Fanuc KAREL source: MP0112.compact.KL

PROGRAM MP0112
%STACKSIZE=65535
%PRIORITY=65535
%NOLOCKGROUP
ROUTINE FINT(P1 : INTEGER) : INTEGER FROM MP0112
ROUTINE FREAL(P1 : REAL) : REAL FROM MP0112
ROUTINE RTEST(P1 : INTEGER; P2 : REAL) FROM MP0112
ROUTINE FINT
BEGIN
RETURN((P1 + 1))
END FINT
ROUTINE FREAL
BEGIN
RETURN((P1 + 1.0))
END FREAL
ROUTINE RTEST
VAR
L1 : XYZWPR
U2C_9 : INTEGER
U2C_10 : INTEGER
U2C_11 : INTEGER
U2C_12 : REAL
U2C_13 : REAL
U2C_14 : REAL
U2C_15 : REAL
S1 : REAL
BEGIN
U2C_9=7
U2C_10=3
U2C_11=2
U2C_12=2.5
U2C_13=4.5
U2C_14=1.5
S1=(L1.X / U2C_13)
END RTEST
BEGIN
RTEST(7,2.5)
END MP0112
